(* Schneider Machine Expert - Basic project 3. Memory Config, file version 2.9.0.0 *)
(* ProjectInformations: Name=New project *)

HARDWARE
  Cpu 0: TM221C24R
  EthernetConfiguration: NetworkName=M221, IpAllocationMode=FixedAddress, IpAddress=0.0.0.0, SubnetMask=0.0.0.0
  SerialLineConfiguration: Baud=Baud19200, Parity=ParityEven, DataBits=DataBits8, StopBits=StopBits1, PhysicalMedium=PhysicalMediumRs485, SlaveId=1, Addressing=SlaveAddressing
  MastTask: UsePeriodScanMode=false, PeriodScan=100
  FastTask: Period=255
  CpuBehavior: StartingMode=StartAsPreviousState, AutoSaveRamOnEeprom=true, WatchdogPeriod=250

SYMBOLS  (address, symbol, comment, settings)
  %M0       MEMORY_1
  %M1       MEMEORY_2
  %I0.0     INPUT_1
  %Q0.0     OUTPUT_1
  %Q0.1     OUTPUT_2

POU New POU
  (* SectionNumber=1 *)

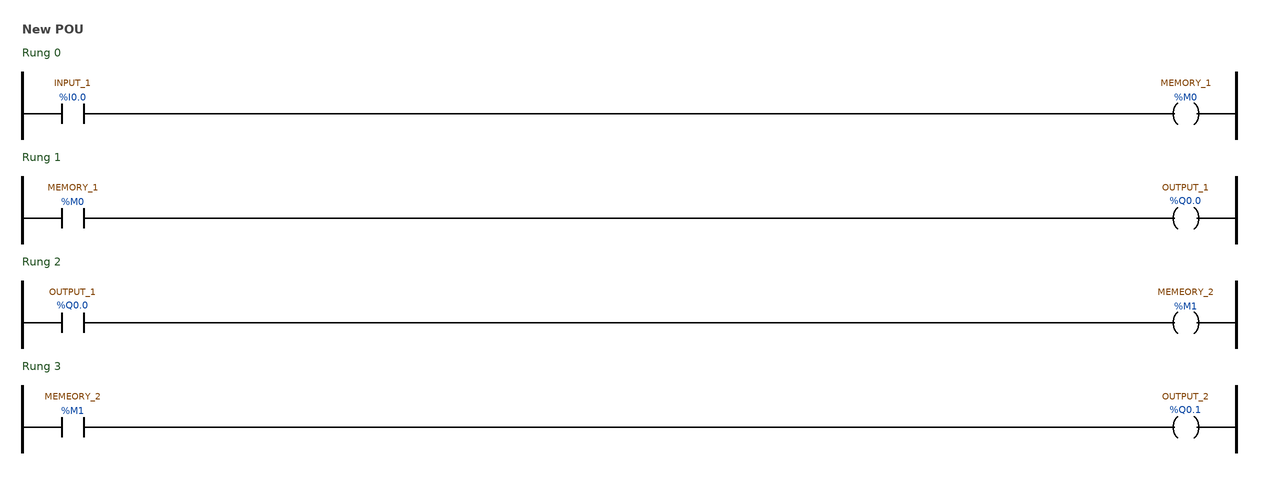

// Rung 0
  LD %I0.0                (* INPUT_1 *)
  ST %M0                  (* MEMORY_1 *)
  // as ST:
  //   MEMORY_1 := INPUT_1;

// Rung 1
  LD %M0                  (* MEMORY_1 *)
  ST %Q0.0                (* OUTPUT_1 *)
  // as ST:
  //   OUTPUT_1 := MEMORY_1;

// Rung 2
  LD %Q0.0                (* OUTPUT_1 *)
  ST %M1                  (* MEMEORY_2 *)
  // as ST:
  //   MEMEORY_2 := OUTPUT_1;

// Rung 3
  LD %M1                  (* MEMEORY_2 *)
  ST %Q0.1                (* OUTPUT_2 *)
  // as ST:
  //   OUTPUT_2 := MEMEORY_2;
